// Mitsubishi GX Works2 project: off타이머   PLC: Q02/Q02H

PROGRAM MAIN
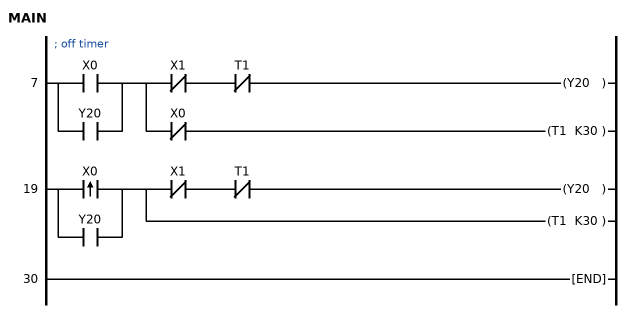
; off timer
7     LD      X0
      OR      Y20
      MPS
      ANI     X1
      ANI     T1
      OUT     Y20
      MPP
      ANI     X0
      OUT     T1 K30
19    LDP     X0
      OR      Y20
      MPS
      ANI     X1
      ANI     T1
      OUT     Y20
      MPP
      OUT     T1 K30
30    END
END_PROGRAM
